TYPE SlotMaterialData EXTENDS SlotHeader :
STRUCT
END_STRUCT
END_TYPE

(* stored: Version 1.1.0.1, ProductVersion 3.1.4020.12
   DUT SlotMaterialData: Id {fcd9b640-f374-4b41-a8a1-cfbe0a8884c8} *)
